TYPE csp_transfer_crosspusher_reject_sensor_status_enum :
(		
	CSP_TRANSFER_CROSSPUSHER_REJECT_SENSOR_STATUS_WAITING						:= 0,
	CSP_TRANSFER_CROSSPUSHER_REJECT_SENSOR_STATUS_START							:= 5,
	CSP_TRANSFER_CROSSPUSHER_REJECT_SENSOR_STATUS_CHECK_PRESENCE_IN_CHUTE		:= 10, 
	CSP_TRANSFER_CROSSPUSHER_REJECT_SENSOR_STATUS_EXTEND_PLATE					:= 20,
	CSP_TRANSFER_CROSSPUSHER_REJECT_SENSOR_STATUS_VERIFY_REJECT					:= 30,
	CSP_TRANSFER_CROSSPUSHER_REJECT_SENSOR_STATUS_RETRACT_PLATE					:= 40,
	CSP_TRANSFER_CROSSPUSHER_REJECT_SENSOR_STATUS_WAIT_RESET					:= 50,
	CSP_TRANSFER_CROSSPUSHER_REJECT_SENSOR_STATUS_DONE							:= 900
) := CSP_TRANSFER_CROSSPUSHER_REJECT_SENSOR_STATUS_WAITING;
END_TYPE

(* stored: Version 1.1.0.1, ProductVersion 3.1.4024.3
   DUT csp_transfer_crosspusher_reject_sensor_status_enum: Id {ab2f3218-6b24-033a-365a-6b0442716280} *)
